(* IEC 61131-3 sources: pandora/pandora/aws-platform-main/aws-platform-main/src/WeldSystem/PowerSources, 5 files *)

(* ---- Pab.st ---- *)
USING Esab.Io;

NAMESPACE Esab.WeldSystem.PowerSources
    TYPE
        {S7.Extern=ReadWrite}
        PabData : STRUCT
            Input : PabToController;
            Output : ControllerToPab;
        END_STRUCT;

        // --- Interface struct declarations
        {S7.Extern=ReadWrite}
        PabToController : STRUCT
            /// Indicates that the Weld On command has been received.
            WeldStarted : DigitalInput;
            /// Set as soon as the welding requirements are met.
            Welding : DigitalInput;
            /// Indicates that the weld is finished. Only applicable for LAF/TAF.
            WeldingFinished : DigitalInput;
            /// TRUE when there is an error present that prohibits start.
            Error : DigitalInput;
            /// TRUE when it is possible to start a weld.
            ReadyToStart : DigitalInput;
            /// Indicates the currently selected weld method. TRUE = AC, FALSE = DC. Aristo 1000 only.
            WeldMethod : DigitalInput;
            /// Set when event information is available. Only set for ~5 seconds and then reset.
            Event : DigitalInput;
            /// Set when import or export function is active.
            FileBusy : DigitalInput;
            /// FALSE = Not coupled, TRUE = Coupled. If this is set the power source is master and has found its parallel slave(s).
            ParallelCoupleStatus : DigitalInput;
            /// The total number of errors or events detected. This equals the number of the last post in the error/event log.
            NumberOfErrors : UIntInput := (Endianness := Endianness#Big);
            /// Requested travel speed (cm/min).
            RequestedTravelSpeed : IntInput := (Endianness := Endianness#Little);
            /// The measured welding voltage.
            MeasuredVoltage : RealInput := (Endianness := Endianness#Little, Scale := REAL#0.1);
            /// The measured welding current.
            MeasuredCurrent : UIntInput := (Endianness := Endianness#Little);
            /// Measured wire speed (cm/min).
            MeasuredWireSpeed : IntInput := (Endianness := Endianness#Little);
            /// Measured travel speed (cm/min).
            MeasuredTravelSpeed : IntInput := (Endianness := Endianness#Little);
            /// The measured heat input.
            MeasuredHeatInput : RealInput := (Endianness := Endianness#Little, Scale := REAL#0.1);
            /// The currently set weld method. Aristo 1000 only.
            SetWeldMethod : UIntInput := (Endianness := Endianness#Big);
            /// The currently set regulation type. Aristo 1000 only.
            SetRegulationType : UIntInput := (Endianness := Endianness#Big);
            /// The AC frequency setpoint. Aristo 1000 only.
            SetAcFrequency : UIntInput := (Endianness := Endianness#Little);
            /// The AC balance setpoint. Aristo 1000 only.
            SetAcBalance : UIntInput := (Endianness := Endianness#Little);
            /// The voltage setpoint.
            SetVoltage : RealInput := (Endianness := Endianness#Little, Scale := REAL#0.1);
            /// The current setpoint.
            SetCurrent : UIntInput := (Endianness := Endianness#Little);
            /// Current wire speed setpoint (cm/min).
            SetWireSpeed : UIntInput := (Endianness := Endianness#Little);
            /// Current travel speed setpoint (cm/min).
            SetTravelSpeed : UIntInput := (Endianness := Endianness#Little);
            /// The current AC offset value.
            SetAcOffset : RealInput := (Endianness := Endianness#Little, Scale := REAL#0.1);
            /// The current AC phase shift value.
            SetAcPhaseShift : UIntInput := (Endianness := Endianness#Little);
            /// Requested wire speed (cm/min).
            RequestedWireSpeed : IntInput := (Endianness := Endianness#Little);
            /// Current weld data set
            SetWeldDataSet : UIntInput := (Endianness := Endianness#Little);
            ErrorEvent : ErrorEvent;
            /// Incremented at 2 Hz, when this value is incrementing the PAB can be considered alive and ready for communication.
            Heartbeat : UIntInput := (Endianness := Endianness#Little);
            /// The current start adjust value in %.
            SetStartAdjust : UIntInput := (Endianness := Endianness#Little);
            /// The current regulation dynamics value.
            SetRegulationDynamics : UIntInput := (Endianness := Endianness#Little);
            /// The current regulation inductance value.
            SetRegulationInductance : UIntInput := (Endianness := Endianness#Little);
        END_STRUCT;

        {S7.Extern=ReadWrite}
        ErrorEvent : STRUCT
            Code : WordInput := (Endianness := Endianness#Little);
            SubCode : UIntInput := (Endianness := Endianness#Big);
            NodeId : UIntInput := (Endianness := Endianness#Big);
            DeviceType : UIntInput := (Endianness := Endianness#Big);
            SubUnit : UIntInput := (Endianness := Endianness#Big);
        END_STRUCT;

        {S7.Extern=ReadWrite}
        ControllerToPab : STRUCT
            Common : PabInputCommon;
            InputArea : ARRAY[1..2] OF PabInputArea;
        END_STRUCT;

        {S7.Extern=ReadWrite}
        PabInputCommon : STRUCT
            /// Starts the weld when set to TRUE, to stop welding set this to FALSE.
            WeldOn : DigitalOutput;
            /// When this is set to TRUE the weld system will perform a quick stop (stopping without doing crater fill).
            QuickStop : DigitalOutput;
            /// Set to TRUE to jog the wire feed in the positive direction (down)
            WireFeedJogPos : DigitalOutput;
            /// Set to TRUE to jog the wire feed in the negative direction (up)
            WireFeedJogNeg : DigitalOutput;
            /// Set to TRUE to jog the travel axis in the positive direction
            TravelAxisJogPos : DigitalOutput;
            /// Set to TRUE to jog the travel axis in the negative direction
            TravelAxisJogNeg : DigitalOutput;
            /// Set to TRUE to jog the ICE wire feed in the positive direction (down)
            IceWireFeedJogPos : DigitalOutput;
            /// Set to TRUE to jog the ICE wire feed in the negative direction (up)
            IceWireFeedJogNeg : DigitalOutput;
            /// High speed (jogging)
            HighSpeed : DigitalOutput;
            /// Switches the active input area (0 = Input area #1, 1 = Input area #2)
            InputAreaSwitch : DigitalOutput;
            /// OPTIONAL! A heartbeat used to tell the PAB that the Controller is alive and well.
            Heartbeat : UIntOutput := (Endianness := Endianness#Big);
        END_STRUCT;

        {S7.Extern=ReadWrite}
        PabInputArea : STRUCT
            /// The weld method.
            WeldMethod : UIntOutput := (Endianness := Endianness#Big);
            /// The regulation type.
            RegulationType : UIntOutput := (Endianness := Endianness#Big);
            /// Weld voltage setpoint.
            Voltage : RealOutput := (Endianness := Endianness#Little, Scale := REAL#0.1);
            /// Wire speed setpoint (cm/min)
            WireSpeed : UIntOutput := (Endianness := Endianness#Little);
            /// Weld current setpoint
            Current : UIntOutput := (Endianness := Endianness#Little);
            /// Travel speed setpoint (cm/min)
            TravelSpeed : UIntOutput := (Endianness := Endianness#Little);
            /// AC frequency setpoint. Aristo 1000 only.
            AcFrequency : UIntOutput := (Endianness := Endianness#Little);
            /// AC balance setpoint. Aristo 1000 only
            AcBalance : UIntOutput := (Endianness := Endianness#Little);
            /// AC offset setpoint. Aristo 1000 only.
            AcOffset : RealOutput := (Endianness := Endianness#Little, Scale := REAL#0.1);
            /// AC phase shift setpoint. Aristo 1000 only
            AcPhaseShift : UIntOutput := (Endianness := Endianness#Little);
            /// Start adjust setpoint in %.
            StartAdjust : UIntOutput := (Endianness := Endianness#Little);
            /// Regulation dynamics setpoint.
            RegulationDynamics : UIntOutput := (Endianness := Endianness#Little);
            /// Regulation inductance setpoint.
            RegulationInductance : UIntOutput := (Endianness := Endianness#Little);
            /// ICE wire speed percentage.
            IceWireSpeedPercentage : UIntOutput := (Endianness := Endianness#Little);
        END_STRUCT;

        /// An enum representing the weld method
        WeldMethod : BYTE (
            DCp := BYTE#0,
            AC := BYTE#1,
            DCn := BYTE#2
        );

        RegulationType : BYTE (
            ConstantAmperage := BYTE#0,
            ConstantWire := BYTE#1,
            ConstantCurrent := BYTE#2
        );

        // --- I/O struct declarations
        {S7.Extern=ReadWrite}
        RawPabToController : STRUCT
            WeldStarted AT %X0.0 : BOOL;
            Welding AT %X0.1 : BOOL;
            WeldingFinished AT %X0.2 : BOOL;
            Error AT %X0.3 : BOOL;
            ReadyToStart AT %X1.3 : BOOL;
            WeldMethod AT %X2.2 : BOOL;
            Event AT %X2.4 : BOOL;
            FileBusy AT %X2.5 : BOOL;
            ParallelCoupleStatus AT %X2.7 : BOOL;
            NumberOfErrors AT %B4 : BYTE;
            RequestedTravelSpeed AT %B6 : INT;
            MeasuredVoltage AT %B8 : INT;
            MeasuredCurrent AT %B10 : UINT;
            MeasuredHeatInput AT %B12 : INT;
            MeasuredWireSpeed AT %B14 : INT;
            MeasuredTravelSpeed AT %B16 : INT;
            SetWeldMethod AT %B18 : BYTE;
            SetRegulationType AT %B19 : BYTE;
            SetAcFrequency AT %B20 : UINT;
            SetAcBalance AT %B22 : UINT;
            SetVoltage AT %B24 : UINT;
            SetCurrent AT %B26 : UINT;
            SetWireSpeed AT %B28 : UINT;
            SetTravelSpeed AT %B30 : UINT;
            SetAcOffset AT %B32 : INT;
            SetWeldDataSet AT %B34 : BYTE;
            SetAcPhaseShift AT %B36 : UINT;
            RequestedWireSpeed AT %B38 : INT;
            ErrorEvent AT %B40 : RawErrorEvent;
            Heartbeat AT %B46 : UINT;
            SetStartAdjust AT %B48 : UINT;
            SetRegulationDynamics AT %B50 : UINT;
            SetRegulationInductance AT %B52 : UINT;
        END_STRUCT;

        {S7.Extern=ReadWrite}
        RawErrorEvent : STRUCT
            Code AT %B0 : WORD;
            SubCode AT %B2 : BYTE;
            NodeId AT %B3 : BYTE;
            DeviceType AT %B4 : BYTE;
            SubUnit AT %B5 : BYTE;
        END_STRUCT;

        {S7.Extern=ReadWrite}
        RawControllerToPab : STRUCT
            Common AT %B0 : RawPabInputCommon;
            Area1 AT %B8 : RawPabInputArea;
            Area2 AT %B36 : RawPabInputArea;
        END_STRUCT;

        {S7.Extern=ReadWrite}
        RawPabInputCommon : STRUCT
            WeldOn AT %X0.0 : BOOL;
            QuickStop AT %X0.1 : BOOL;
            WireFeedJogPos AT %X0.4 : BOOL;
            WireFeedJogNeg AT %X0.5 : BOOL;
            TravelAxisJogPos AT %X0.6 : BOOL;
            TravelAxisJogNeg AT %X0.7 : BOOL;
            IceWireFeedJogPos AT %X1.0 : BOOL;
            IceWireFeedJogNeg AT %X1.1 : BOOL;
            HighSpeed AT %X1.2 : BOOL;
            InputAreaSwitch AT %X3.2 : BOOL;
            Heartbeat AT %B7 : BYTE;
        END_STRUCT;

        {S7.Extern=ReadWrite}
        RawPabInputArea : STRUCT
            WeldMethod AT %B0 : BYTE;
            RegulationType AT %B1 : BYTE;
            Voltage AT %B2 : UINT;
            WireSpeed AT %B4 : UINT;
            Current AT %B6 : UINT;
            TravelSpeed AT %B8 : UINT;
            AcFrequency AT %B10 : UINT;
            AcBalance AT %B12 : UINT;
            AcOffset AT %B14 : INT;
            AcPhaseShift AT %B16 : UINT;
            StartAdjust AT %B18 : UINT;
            RegulationDynamics AT %B20 : UINT;
            RegulationInductance AT %B22 : UINT;
            IceWireSpeedPercentage AT %B26 : UINT;
        END_STRUCT;
    END_TYPE

    FUNCTION PabRead
        VAR_INPUT
            Processed : REF_TO PabToController;
            Raw : REF_TO RawPabToController;
        END_VAR

        Processed^.WeldStarted.Read             (Raw^.WeldStarted);
        Processed^.Welding.Read                 (Raw^.Welding);
        Processed^.WeldingFinished.Read         (Raw^.WeldingFinished);
        Processed^.Error.Read                   (Raw^.Error);
        Processed^.ReadyToStart.Read            (Raw^.ReadyToStart);
        Processed^.WeldMethod.Read              (Raw^.WeldMethod);
        Processed^.Event.Read                   (Raw^.Event);
        Processed^.FileBusy.Read                (Raw^.FileBusy);
        Processed^.ParallelCoupleStatus.Read    (Raw^.ParallelCoupleStatus);
        Processed^.NumberOfErrors.Read          (Raw^.NumberOfErrors);
        Processed^.RequestedTravelSpeed.Read    (Raw^.RequestedTravelSpeed);
        Processed^.MeasuredVoltage.Read         (Raw^.MeasuredVoltage);
        Processed^.MeasuredCurrent.Read         (Raw^.MeasuredCurrent);
        Processed^.MeasuredHeatInput.Read       (Raw^.MeasuredHeatInput);
        Processed^.MeasuredWireSpeed.Read       (Raw^.MeasuredWireSpeed);
        Processed^.MeasuredTravelSpeed.Read     (Raw^.MeasuredTravelSpeed);
        Processed^.SetWeldMethod.Read           (Raw^.SetWeldMethod);
        Processed^.SetRegulationType.Read       (Raw^.SetRegulationType);
        Processed^.SetAcFrequency.Read          (Raw^.SetAcFrequency);
        Processed^.SetAcBalance.Read            (Raw^.SetAcBalance);
        Processed^.SetVoltage.Read              (Raw^.SetVoltage);
        Processed^.SetCurrent.Read              (Raw^.SetCurrent);
        Processed^.SetWireSpeed.Read            (Raw^.SetWireSpeed);
        Processed^.SetTravelSpeed.Read          (Raw^.SetTravelSpeed);
        Processed^.SetAcOffset.Read             (Raw^.SetAcOffset);
        Processed^.SetWeldDataSet.Read          (Raw^.SetWeldDataSet);
        Processed^.SetAcPhaseShift.Read         (Raw^.SetAcPhaseShift);
        Processed^.RequestedWireSpeed.Read      (Raw^.RequestedWireSpeed);
        Processed^.ErrorEvent.Code.Read         (Raw^.ErrorEvent.Code);
        Processed^.ErrorEvent.SubCode.Read      (Raw^.ErrorEvent.SubCode);
        Processed^.ErrorEvent.NodeId.Read       (Raw^.ErrorEvent.NodeId);
        Processed^.ErrorEvent.DeviceType.Read   (Raw^.ErrorEvent.DeviceType);
        Processed^.ErrorEvent.SubUnit.Read      (Raw^.ErrorEvent.SubUnit);
        Processed^.Heartbeat.Read               (Raw^.Heartbeat);
        Processed^.SetStartAdjust.Read          (Raw^.SetStartAdjust);
        Processed^.SetRegulationDynamics.Read   (Raw^.SetRegulationDynamics);
        Processed^.SetRegulationInductance.Read (Raw^.SetRegulationInductance);
    END_FUNCTION

    FUNCTION PabWrite
        VAR_INPUT
            Processed : REF_TO ControllerToPab;
            Raw : REF_TO RawControllerToPab;
        END_VAR

        Processed^.Common.WeldOn.Write              (Raw^.Common.WeldOn);
        Processed^.Common.QuickStop.Write           (Raw^.Common.QuickStop);
        Processed^.Common.Heartbeat.Write           (Raw^.Common.Heartbeat);
        Processed^.Common.WireFeedJogPos.Write      (Raw^.Common.WireFeedJogPos);
        Processed^.Common.WireFeedJogNeg.Write      (Raw^.Common.WireFeedJogNeg);
        Processed^.Common.TravelAxisJogPos.Write    (Raw^.Common.TravelAxisJogPos);
        Processed^.Common.TravelAxisJogNeg.Write    (Raw^.Common.TravelAxisJogNeg);
        Processed^.Common.IceWireFeedJogPos.Write   (Raw^.Common.IceWireFeedJogPos);
        Processed^.Common.IceWireFeedJogNeg.Write   (Raw^.Common.IceWireFeedJogNeg);
        Processed^.Common.HighSpeed.Write           (Raw^.Common.HighSpeed);
        Processed^.Common.InputAreaSwitch.Write     (Raw^.Common.InputAreaSwitch);

        Processed^.InputArea[1].WeldMethod.Write               (Raw^.Area1.WeldMethod);
        Processed^.InputArea[1].RegulationType.Write           (Raw^.Area1.RegulationType);
        Processed^.InputArea[1].Voltage.Write                  (Raw^.Area1.Voltage);
        Processed^.InputArea[1].WireSpeed.Write                (Raw^.Area1.WireSpeed);
        Processed^.InputArea[1].Current.Write                  (Raw^.Area1.Current);
        Processed^.InputArea[1].TravelSpeed.Write              (Raw^.Area1.TravelSpeed);
        Processed^.InputArea[1].AcFrequency.Write              (Raw^.Area1.AcFrequency);
        Processed^.InputArea[1].AcBalance.Write                (Raw^.Area1.AcBalance);
        Processed^.InputArea[1].AcOffset.Write                 (Raw^.Area1.AcOffset);
        Processed^.InputArea[1].AcPhaseShift.Write             (Raw^.Area1.AcPhaseShift);
        Processed^.InputArea[1].StartAdjust.Write              (Raw^.Area1.StartAdjust);
        Processed^.InputArea[1].RegulationDynamics.Write       (Raw^.Area1.RegulationDynamics);
        Processed^.InputArea[1].RegulationInductance.Write     (Raw^.Area1.RegulationInductance);
        Processed^.InputArea[1].IceWireSpeedPercentage.Write   (Raw^.Area1.IceWireSpeedPercentage);

        Processed^.InputArea[2].WeldMethod.Write               (Raw^.Area2.WeldMethod);
        Processed^.InputArea[2].RegulationType.Write           (Raw^.Area2.RegulationType);
        Processed^.InputArea[2].Voltage.Write                  (Raw^.Area2.Voltage);
        Processed^.InputArea[2].WireSpeed.Write                (Raw^.Area2.WireSpeed);
        Processed^.InputArea[2].Current.Write                  (Raw^.Area2.Current);
        Processed^.InputArea[2].TravelSpeed.Write              (Raw^.Area2.TravelSpeed);
        Processed^.InputArea[2].AcFrequency.Write              (Raw^.Area2.AcFrequency);
        Processed^.InputArea[2].AcBalance.Write                (Raw^.Area2.AcBalance);
        Processed^.InputArea[2].AcOffset.Write                 (Raw^.Area2.AcOffset);
        Processed^.InputArea[2].AcPhaseShift.Write             (Raw^.Area2.AcPhaseShift);
        Processed^.InputArea[2].StartAdjust.Write              (Raw^.Area2.StartAdjust);
        Processed^.InputArea[2].RegulationDynamics.Write       (Raw^.Area2.RegulationDynamics);
        Processed^.InputArea[2].RegulationInductance.Write     (Raw^.Area2.RegulationInductance);
        Processed^.InputArea[2].IceWireSpeedPercentage.Write   (Raw^.Area2.IceWireSpeedPercentage);
    END_FUNCTION

END_NAMESPACE

(* ---- PowerSource.st ---- *)
USING Esab.Utils.Assets;
USING Esab.Utils.Timer;
USING Esab.Utils.Io;

USING Esab.WeldSystem;

USING System.FastMath;

NAMESPACE Esab.WeldSystem.PowerSources

    INTERFACE IPowerSource
        /// Intended for cyclic execution
        METHOD Execute
        END_METHOD

        /// Sets a listener to this power source
        METHOD SetListener
            VAR_INPUT
                listener : IPowerSourceListener;
            END_VAR
        END_METHOD

        /// Initiates the welding sequence
        METHOD Start
        END_METHOD

        /// Stops the welding sequence in a controlled manner
        METHOD Stop
        END_METHOD

        /// Stops the welding sequence faster, skips the stop phase
        METHOD QuickStop
        END_METHOD

        /// Sets remote start towards the power source
        METHOD RemoteStart
        END_METHOD

        /// Sets remote stop towards the power source
        METHOD RemoteStop
        END_METHOD

        /// Returns a reference to the currently active input area
        METHOD ActiveArea : REF_TO SetPoints
        END_METHOD

        /// Returns a reference to the currently passive input area
        METHOD PassiveArea : REF_TO SetPoints
        END_METHOD

        /// Switch the active and passive areas
        METHOD SwitchActivePassive
        END_METHOD

        /// Sets the travel control (NOTE: Async)
        METHOD SetTravelControl
            VAR_INPUT
                control : TravelControl;
            END_VAR
        END_METHOD

        /// Sets the travel motor drive (NOTE: Async)
        METHOD SetTravelMotorDrive
            VAR_INPUT
                drive : TravelMotorDrive;
            END_VAR
        END_METHOD

        /// Sets the tandem role of this power source (NOTE: Async)
        METHOD SetTandemRole
            VAR_INPUT
                role : TandemRole;
            END_VAR
        END_METHOD

        /// Sets the start type (NOTE: Async)
        METHOD SetStartType
            VAR_INPUT
                startType : StartType;
            END_VAR
        END_METHOD

        /// Sets normal wire feed jog speed (NOTE: Async)
        METHOD SetWireFeedJogSpeed
            VAR_INPUT
                speed : UINT;
            END_VAR
        END_METHOD

        /// Sets wire feed jog high speed (NOTE: Async)
        METHOD SetWireFeedJogHighSpeed
            VAR_INPUT
                speed : UINT;
            END_VAR
        END_METHOD

        /// Applies a configuration to the wire motor
        /// Returns FALSE if it is not currently possible to set configuration
        METHOD ApplyWireMotorConfiguration : BOOL
            VAR_INPUT
                motorConfiguration : REF_TO MotorConfiguration;
            END_VAR
        END_METHOD

        /// ID of the power source
        METHOD GetId : UINT
        END_METHOD

        /// Node ID used by this power source
        METHOD GetNodeId : UINT
        END_METHOD

        /// The actual weld system type that is connected
        METHOD GetWeldSystemType : WeldSystemType
        END_METHOD

        /// Travel control (Off/Enabled)
        METHOD GetTravelControl : TravelControl
        END_METHOD

        /// Travel motor drive (Faa/External)
        METHOD GetTravelMotorDrive : TravelMotorDrive
        END_METHOD

        /// Tandem role (Head/Tail)
        METHOD GetTandemRole : TandemRole
        END_METHOD

        /// Returns TRUE if the welding system is welding
        METHOD IsWelding : BOOL
        END_METHOD

        /// Returns TRUE if the PLC has active communication with the PAB
        METHOD IsConnected : BOOL
        END_METHOD

        /// Returns TRUE if the power source reports as ready to start
        METHOD IsReadyToStart : BOOL
        END_METHOD

        /// Returns TRUE if the power source reports it has an error
        METHOD HasError : BOOL
        END_METHOD

        /// Returns the measured welding voltage.
        METHOD GetMeasuredVoltage : REAL
        END_METHOD

        /// Returns the measured wire speed (cm/min)
        METHOD GetMeasuredWireSpeed : INT
        END_METHOD

        /// Returns the measured travel speed (cm/min)
        METHOD GetMeasuredTravelSpeed : INT
        END_METHOD

        /// Returns the measured heat input (kJ/cm)
        METHOD GetMeasuredHeatInput : REAL
        END_METHOD

        /// Returns the currently set weld data set
        METHOD GetWeldDataSet : UINT
        END_METHOD

        /// Returns the requested (by the power source) travel speed
        METHOD GetRequestedTravelSpeed : INT
        END_METHOD

        /// Returns the requested (by the power source) wire speed
        METHOD GetRequestedWireSpeed : INT
        END_METHOD

        /// Returns TRUE if the node with the given ID is connected
        METHOD NodeIsConnected : BOOL
            VAR_INPUT
                nodeId : UINT;
            END_VAR
        END_METHOD

        /// Returns the information of the given node
        METHOD GetNodeInformation : NodeInformation
            VAR_INPUT
                nodeId : UINT;
            END_VAR
        END_METHOD

        METHOD WireFeedJogPos
            VAR_INPUT
                highSpeed : BOOL;
            END_VAR
        END_METHOD

        METHOD WireFeedJogNeg
            VAR_INPUT
                highSpeed : BOOL;
            END_VAR
        END_METHOD

        METHOD TravelAxisJogPos
            VAR_INPUT
                highSpeed : BOOL;
            END_VAR
        END_METHOD

        METHOD TravelAxisJogNeg
            VAR_INPUT
                highSpeed : BOOL;
            END_VAR
        END_METHOD

        /// Initiates a read of all connected nodes (unless already reading)
        METHOD ReadNodes
        END_METHOD

        METHOD WriteAsync
            VAR_INPUT
                record : DataRecord;
                value : UINT;
            END_VAR
        END_METHOD

        METHOD WriteAsync
            VAR_INPUT
                command: REF_TO UIntAsyncCommand;
            END_VAR
        END_METHOD

        METHOD ReadAsync
            VAR_INPUT
                record : DataRecord;
            END_VAR
        END_METHOD

        METHOD ReadAsync
            VAR_INPUT
                command: REF_TO UIntAsyncCommand;
            END_VAR
        END_METHOD
    END_INTERFACE

    INTERFACE IHeartBeat
        /// Returns TRUE if this object is initialized
        METHOD IsInitialized : BOOL
        END_METHOD

        /// Cyclic execution to evaluate heartbeat
        METHOD Execute
        END_METHOD

        /// Returns TRUE if a heartbeat is detected
        METHOD Alive : BOOL
        END_METHOD

        /// Returns TRUE if no heartbeat is detected
        METHOD Dead : BOOL
        END_METHOD
    END_INTERFACE

    CLASS Heartbeat IMPLEMENTS IHeartbeat
        VAR PUBLIC
            Input : IUIntInput;
            Timer: ITimer;
        END_VAR

        VAR PRIVATE
            _value : UINT;
            _lastValue : UINT;
            _alive : BOOL;
        END_VAR

        METHOD PUBLIC IsInitialized : BOOL
            IsInitialized := Input <> NULL AND Timer <> NULL;
        END_METHOD

        METHOD PUBLIC Execute
            IF NOT THIS.IsInitialized() THEN
                _alive := FALSE;
                RETURN;
            END_IF;

            _lastValue := _value;
            _value := Input.GetValue();

            Timer.Execute(_value = _lastValue, LT#10s);
            _alive := NOT Timer.Expired();
        END_METHOD

        METHOD PUBLIC Alive : BOOL
            Alive := _alive;
        END_METHOD

        METHOD PUBLIC Dead : BOOL
            Dead := NOT _alive;
        END_METHOD
    END_CLASS

    INTERFACE IPowerSourceListener
        /// Called when a power source becomes connected
        METHOD PowerSourceConnected
            VAR_INPUT
                /// The id (enumeration) of the power source
                id : UINT;
            END_VAR
        END_METHOD

        /// Called when a power source disconnects
        METHOD PowerSourceDisconnected
            VAR_INPUT
                /// The id (enumeration) of the power source
                id : UINT;
            END_VAR
        END_METHOD
    END_INTERFACE

    TYPE
        WeldProcess : INT(
            Saw := 0,
            Gmaw := 1,
            Gouging := 2
        );

        WireType : INT(
            FeSolidSingle := 0,
            FeSolidTwin := 1,
            FeTubeSingle := 2,
            FeTubeTwin := 3,
            SsSolidSingle := 4,
            SsSolidTwin := 5,
            SsTubeSingle := 6,
            SsTubeTwin := 7,
            AlSolidSingle := 8,
            AlSolidTwin := 9,
            StripSingle := 10,
            Gouging := 11
        );

        StartType : INT(
            Direct := 0,
            Scratch := 1,
            Lwas := 2,
            LwasMan := 3
        );

        TravelControl : INT(
            Off := 0,
            Enabled := 1
        );

        TravelMotorDrive : INT(
            Faa := 0,
            External := 1
        );

        TandemRole : INT(
            Head := 0,
            Slave := 1
        );

        /// Container for values read from async commands
        StatusBuffer : STRUCT
            /// Node ID used by this power source
            NodeId : UINT;
            /// The actual weld system type that is connected
            WeldSystemType : WeldSystemType;
            /// Travel control (Off/Enabled)
            TravelControl : TravelControl;
            /// Travel motor drive (Faa/External)
            TravelMotorDrive : TravelMotorDrive;
            /// Tandem role (Head/Tail)
            TandemRole : TandemRole;
        END_STRUCT;
    END_TYPE

    CLASS PowerSourceObservable IMPLEMENTS IAssetObservable
        VAR PUBLIC
            State : PowerSourceState;
            ReadyToStart : BOOL;
            Welding : BOOL;
            Error : BOOL;
            Connected : BOOL;
            WeldMethod : WeldMethod;
            MeasuredVoltage : REAL;
            MeasuredCurrent : UINT;
            MeasuredHeatInput : REAL;
            MeasuredWireSpeed : INT;
            MeasuredTravelSpeed : INT;
            RequestedWireSpeed : INT;
            RequestedTravelSpeed : INT;
            SetPoints : SetPoints;
        END_VAR
    END_CLASS

    FUNCTION CalculateMotorScaleFactors
        VAR_INPUT
            motorConfiguration : REF_TO MotorConfiguration;
        END_VAR

        VAR_OUTPUT
            nominator : UINT;
            denominator : UINT;
        END_VAR

        nominator := TO_UINT(TO_LREAL(motorConfiguration^.Gear.N2) / motorConfiguration^.Gear.N1 * motorConfiguration^.Rpm * motorConfiguration^.FeedRollDiameter * Constants#PI);
        denominator := TO_UINT(TO_UDINT(motorConfiguration^.Rpm) * motorConfiguration^.EncoderPpr / UINT#60);
    END_FUNCTION

    TYPE
        {S7.Extern=ReadWrite}
        RuntimeParameters : STRUCT
            WireFeedJogSpeed : UINT;
            WireFeedJogHighSpeed : UINT;
        END_STRUCT;

        {S7.Extern=ReadWrite}
        HardwareConfiguration : STRUCT
            WireMotor : MotorConfiguration;
        END_STRUCT;

        {S7.Extern=ReadWrite}
        MotorConfiguration : STRUCT
            Gear : Gear;
            Rpm : UINT;
            FeedRollDiameter : UINT;
            EncoderPpr : UINT;
            MaxCurrent : UINT;
        END_STRUCT;

        {S7.Extern=ReadWrite}
        Gear : STRUCT
            N1 : UINT;
            N2 : UINT;
        END_STRUCT;

        {S7.Extern=ReadWrite}
        Io : STRUCT
            Pab : PabData;
            Output : Output;
        END_STRUCT;

        {S7.Extern=ReadWrite}
        Output : STRUCT
            RemoteStart : DigitalOutput;
        END_STRUCT;

        PowerSourceState : INT(
            Idle := 0,
            NotConnected := 1,
            Error := 2,
            Welding := 3
        );

        SetPoints : STRUCT
            Voltage : REAL;
            Current : UINT;
            WireSpeed : UINT;
            TravelSpeed : UINT;
            AcFrequency : UINT;
            AcBalance : UINT;
            AcOffset : REAL;
            AcPhaseShift : UINT;
            WeldMethod : WeldMethod;
            RegulationType : RegulationType;
            StartAdjust : UINT;
            RegulationDynamics : UINT;
            RegulationInductance : UINT;
            IceWireSpeedPercentage : UINT;
        END_STRUCT;
    END_TYPE

END_NAMESPACE

(* ---- Aristo1000.st ---- *)
USING Esab.Api;
USING Esab.Utils.Alarming;
USING Esab.Utils;
USING Esab.Utils.Assets;
USING Esab.WeldSystem.PowerSources;
USING Esab.Utils.Alarming;
USING Siemens.Simatic.S71500.Alarming;
USING Siemens.Simatic.S71500.DistributedIO;

NAMESPACE Esab.WeldSystem.PowerSources.Aristo1000

    /// This class implements an Aristo 1000 power source
    CLASS PowerSource EXTENDS Asset IMPLEMENTS IPowerSource, IAsyncCommandListener
        VAR PRIVATE
            _id : UINT;
            _ioDeviceId : WORD;
            _heartbeat: IHeartBeat;
            _io : REF_TO Io;
            _runtimeParameters : REF_TO RuntimeParameters;
            _hardwareConfiguration : REF_TO HardwareConfiguration;
            _asyncInterface : IAsyncInterface;
            _asyncCommands : AsyncCommands;
            _errorAlarm : IAlarm;
            _heartbeatAlarm : IAlarm;
            _asyncCommandReadAlarm : IAlarm;
            _asyncCommandWriteAlarm : IAlarm;
            _asyncCommandNullAlarm : IAlarm;

            _readingNodes : BOOL := FALSE;
            _currentlyReadingNodeId : UINT := UINT#0;
            _nodeInformation : ARRAY [1..31] OF NodeInformation;
            _observable : PowerSourceObservable;
            _listener : IPowerSourceListener := NULL;
            _isConnected : BOOL := FALSE;

            _nodeId : UINT := UINT#0;
            _weldSystemType : WeldSystemType;
            _travelControl : TravelControl;
            _travelMotorDrive : TravelMotorDrive;
            _tandemRole : TandemRole;
            _inputAreaSwitch : BOOL := FALSE; // Area 2 is active if True
            _inputArea : ARRAY [1..2] OF SetPoints;

            // Commands used when reading/writing custom records
            _writeUIntAsyncCommand : UIntAsyncCommand;
            _readUIntAsyncCommand : UIntAsyncCommand;

            _highSpeed : BOOL := FALSE;
            _wireFeedJogPos : BOOL := FALSE;
            _wireFeedJogNeg : BOOL := FALSE;
            _travelAxisJogPos : BOOL := FALSE;
            _travelAxisJogNeg : BOOL := FALSE;
        END_VAR

        METHOD PUBLIC Setup
            VAR_INPUT
                id : UINT;
                ioDeviceId : WORD;
                heartbeat: IHeartBeat;
                io : REF_TO Io;
                runtimeParameters : REF_TO RuntimeParameters;
                hardwareConfiguration : REF_TO HardwareConfiguration;
                asyncInterface : IAsyncInterface;
                errorAlarm : IAlarm;
                heartbeatAlarm : IAlarm;
                asyncCommandReadAlarm : IAlarm;
                asyncCommandWriteAlarm : IAlarm;
                asyncCommandNullAlarm : IAlarm;
                setupAlarm : IAlarm;
            END_VAR

            _id := id;
            _ioDeviceId := ioDeviceId;
            _heartbeat := heartbeat;
            _io := io;
            _runtimeParameters := runtimeParameters;
            _hardwareConfiguration := hardwareConfiguration;
            _asyncInterface := asyncInterface;
            _asyncInterface.SetListener(THIS);
            _errorAlarm := errorAlarm;
            _heartbeatAlarm := heartbeatAlarm;
            _asyncCommandReadAlarm := asyncCommandReadAlarm;
            _asyncCommandWriteAlarm := asyncCommandWriteAlarm;
            _asyncCommandNullAlarm := asyncCommandNullAlarm;
            _setupAlarm := setupAlarm;

            _isSetup := _io <> NULL AND
                        _heartbeat <> NULL AND
                        _runtimeParameters <> NULL AND
                        _hardwareConfiguration <> NULL AND
                        _errorAlarm <> NULL AND
                        _heartbeatAlarm <> NULL AND
                        _asyncCommandReadAlarm <> NULL AND
                        _asyncCommandWriteAlarm <> NULL AND
                        _asyncCommandNullAlarm <> NULL;

            IF _isSetup THEN
                THIS.WriteAsync(DataRecord#WireJogLowSpeed, _runtimeParameters^.WireFeedJogSpeed);
                THIS.WriteAsync(DataRecord#WireJogHighSpeed, _runtimeParameters^.WireFeedJogHighSpeed);
            END_IF;
        END_METHOD

        METHOD PUBLIC OVERRIDE Execute
            SUPER.Execute();

            IF _setupAlarm.IsActive() THEN
                RETURN;
            END_IF;

            _heartbeat.Execute();

            _heartbeatAlarm.Execute(SIG := _heartbeat.Dead());

            IF _heartbeat.Dead() THEN
                IF _isConnected AND _listener <> NULL THEN
                    _listener.PowerSourceDisconnected(THIS.GetId());
                END_IF;

                RETURN;
            ELSIF NOT _isConnected AND _listener <> NULL THEN
                THIS.ReadNodes();
                _listener.PowerSourceConnected(THIS.GetId());
            END_IF;

            _isConnected := _heartbeat.Alive();

            THIS.SetHeartbeat(THIS.GetHeartbeat());

            _errorAlarm.Execute(SIG := _io^.Pab.Input.Error.GetValue());

            _io^.Pab.Output.Common.HighSpeed.SetValue(_highSpeed);
            _io^.Pab.Output.Common.WireFeedJogPos.SetValue(_wireFeedJogPos);
            _io^.Pab.Output.Common.WireFeedJogNeg.SetValue(_wireFeedJogNeg);
            _io^.Pab.Output.Common.TravelAxisJogPos.SetValue(_travelAxisJogPos);
            _io^.Pab.Output.Common.TravelAxisJogNeg.SetValue(_travelAxisJogNeg);

            _highSpeed := FALSE;
            _wireFeedJogPos := FALSE;
            _wireFeedJogNeg := FALSE;
            _travelAxisJogPos := FALSE;
            _travelAxisJogNeg := FALSE;

            IF _io^.Pab.Input.Welding.FallingEdge() THEN
                THIS.Stop();
            END_IF;

            _asyncInterface.Execute();

            THIS.UpdateObservable();
            THIS.UpdateSetpoints();
        END_METHOD

        METHOD PUBLIC OVERRIDE UpdateState
            IF _setupAlarm.IsActive() THEN
                _currentState := PowerSourceState#Error;
            ELSIF NOT THIS.IsConnected() THEN
                _currentState := PowerSourceState#NotConnected;
            ELSIF THIS.IsWelding() THEN
                _currentState := PowerSourceState#Welding;
            ELSIF _errorAlarm.IsActive() OR _asyncCommandReadAlarm.IsActive() OR _asyncCommandWriteAlarm.IsActive() OR _asyncCommandNullAlarm.IsActive() THEN
                _currentState := PowerSourceState#Error;
            ELSE
                _currentState := PowerSourceState#Idle;
            END_IF;
        END_METHOD

        METHOD PUBLIC SetListener
            VAR_INPUT
                listener : IPowerSourceListener;
            END_VAR

            _listener := listener;
        END_METHOD

        METHOD PUBLIC Start
            _io^.Pab.Output.Common.WeldOn.SetValue(TRUE);
        END_METHOD

        METHOD PUBLIC Stop
            _io^.Pab.Output.Common.WeldOn.SetValue(FALSE);
        END_METHOD

        METHOD PUBLIC QuickStop
            _io^.Pab.Output.Common.WeldOn.SetValue(FALSE);
            _io^.Pab.Output.Common.QuickStop.SetValue(TRUE);
        END_METHOD

        METHOD PUBLIC RemoteStart
            _io^.Output.RemoteStart.SetValue(TRUE);
        END_METHOD

        METHOD PUBLIC RemoteStop
            _io^.Output.RemoteStart.SetValue(FALSE);
        END_METHOD

        METHOD PUBLIC ActiveArea : REF_TO SetPoints
            IF NOT _inputAreaSwitch THEN
                ActiveArea := REF(_inputArea[1]);
            ELSE
                ActiveArea := REF(_inputArea[2]);
            END_IF;
        END_METHOD

        METHOD PUBLIC PassiveArea : REF_TO SetPoints
            IF NOT _inputAreaSwitch THEN
                PassiveArea := REF(_inputArea[2]);
            ELSE
                PassiveArea := REF(_inputArea[1]);
            END_IF;
        END_METHOD

        METHOD PUBLIC SwitchActivePassive
            _inputAreaSwitch := NOT _inputAreaSwitch;
            _io^.Pab.Output.Common.InputAreaSwitch.SetValue(_inputAreaSwitch);
        END_METHOD

        METHOD PUBLIC IsWelding : BOOL
            IsWelding := _io^.Pab.Input.Welding.GetValue() OR _io^.Pab.Input.WeldStarted.GetValue();
        END_METHOD

        METHOD PUBLIC IsConnected : BOOL
            IsConnected := _heartbeat.Alive();
        END_METHOD

        METHOD PUBLIC IsReadyToStart : BOOL
            IsReadyToStart := _io^.Pab.Input.ReadyToStart.GetValue();
        END_METHOD

        METHOD PUBLIC HasError : BOOL
            HasError := _io^.Pab.Input.Error.GetValue();
        END_METHOD

        METHOD PUBLIC SetTravelControl
            VAR_INPUT
                control : TravelControl;
            END_VAR

            _travelControl := control;
            _asyncCommands.TravelControl.Value := TO_UINT(control);

            _asyncInterface.WriteCommand(REF(_asyncCommands.TravelControl));
        END_METHOD

        METHOD PUBLIC SetTravelMotorDrive
            VAR_INPUT
                drive : TravelMotorDrive;
            END_VAR

            _travelMotorDrive := drive;
            _asyncCommands.TravelMotorDrive.Value := TO_UINT(drive);

            _asyncInterface.WriteCommand(REF(_asyncCommands.TravelMotorDrive));
        END_METHOD

        METHOD PUBLIC SetTandemRole
            VAR_INPUT
                role : TandemRole;
            END_VAR

            _tandemRole := role;
            _asyncCommands.TandemRole.Value := TO_UINT(role);

            _asyncInterface.WriteCommand(REF(_asyncCommands.TandemRole));
        END_METHOD

        METHOD PUBLIC SetStartType
            VAR_INPUT
                startType : StartType;
            END_VAR

            _asyncCommands.StartType.Value := TO_UINT(startType);

            _asyncInterface.WriteCommand(REF(_asyncCommands.StartType));
        END_METHOD

        METHOD PUBLIC SetWireFeedJogSpeed
            VAR_INPUT
                speed : UINT;
            END_VAR

            _asyncCommands.JogWireFeedSpeed.Value := speed;
            _asyncInterface.WriteCommand(REF(_asyncCommands.JogWireFeedSpeed));
        END_METHOD

        METHOD PUBLIC SetWireFeedJogHighSpeed
            VAR_INPUT
                speed : UINT;
            END_VAR

            _asyncCommands.JogWireFeedHighSpeed.Value := speed;
            _asyncInterface.WriteCommand(REF(_asyncCommands.JogWireFeedHighSpeed));
        END_METHOD

        METHOD PUBLIC GetId : UINT
            GetId := _id;
        END_METHOD

        METHOD PUBLIC GetNodeId : UINT
            GetNodeId := _nodeId;
        END_METHOD

        METHOD PUBLIC GetWeldSystemType : WeldSystemType
            GetWeldSystemType := _weldSystemType;
        END_METHOD

        METHOD PUBLIC GetTravelControl : TravelControl
            GetTravelControl := _travelControl;
        END_METHOD

        METHOD PUBLIC GetTravelMotorDrive : TravelMotorDrive
            GetTravelMotorDrive := _travelMotorDrive;
        END_METHOD

        METHOD PUBLIC GetTandemRole : TandemRole
            GetTandemRole := _tandemRole;
        END_METHOD

        METHOD PUBLIC GetMeasuredVoltage : REAL
            GetMeasuredVoltage := _io^.Pab.Input.MeasuredVoltage.GetValue();
        END_METHOD

        METHOD PUBLIC GetMeasuredCurrent : UINT
            GetMeasuredCurrent := _io^.Pab.Input.MeasuredCurrent.GetValue();
        END_METHOD

        METHOD PUBLIC GetMeasuredWireSpeed : INT
            GetMeasuredWireSpeed := _io^.Pab.Input.MeasuredWireSpeed.GetValue();
        END_METHOD

        METHOD PUBLIC GetMeasuredTravelSpeed : INT
            GetMeasuredTravelSpeed := _io^.Pab.Input.MeasuredTravelSpeed.GetValue();
        END_METHOD

        METHOD PUBLIC GetMeasuredHeatInput : REAL
            GetMeasuredHeatInput := _io^.Pab.Input.MeasuredHeatInput.GetValue();
        END_METHOD

        METHOD PUBLIC GetWeldDataSet : UINT
            GetWeldDataSet := _io^.Pab.Input.SetWeldDataSet.GetValue();
        END_METHOD

        METHOD PUBLIC GetRequestedTravelSpeed : INT
            GetRequestedTravelSpeed := _io^.Pab.Input.RequestedTravelSpeed.GetValue();
        END_METHOD

        METHOD PUBLIC GetRequestedWireSpeed : INT
            GetRequestedWireSpeed := _io^.Pab.Input.RequestedWireSpeed.GetValue();
        END_METHOD

        METHOD PUBLIC WireFeedJogPos
            VAR_INPUT
                highSpeed : BOOL;
            END_VAR

            _highSpeed := highSpeed;
            _wireFeedJogPos := TRUE;
        END_METHOD

        METHOD PUBLIC WireFeedJogNeg
            VAR_INPUT
                highSpeed : BOOL;
            END_VAR

            _highSpeed := highSpeed;
            _wireFeedJogNeg := TRUE;
        END_METHOD

        METHOD PUBLIC TravelAxisJogPos
            VAR_INPUT
                highSpeed : BOOL;
            END_VAR

            _highSpeed := highSpeed;
            _travelAxisJogPos := TRUE;
        END_METHOD

        METHOD PUBLIC TravelAxisJogNeg
            VAR_INPUT
                highSpeed : BOOL;
            END_VAR

            _highSpeed := highSpeed;
            _travelAxisJogNeg := TRUE;
        END_METHOD

        METHOD PUBLIC ReadNodes
            IF _readingNodes = FALSE THEN
                _readingNodes := TRUE;
                _asyncInterface.ReadCommand(REF(_asyncCommands.ConnectedUnits));
            END_IF;
        END_METHOD

        METHOD PUBLIC NodeIsConnected : BOOL
            VAR_INPUT
                nodeId : UINT;
            END_VAR

            NodeIsConnected := _nodeInformation[nodeId].Connected;
        END_METHOD

        METHOD PUBLIC GetNodeInformation : NodeInformation
            VAR_INPUT
                nodeId : UINT;
            END_VAR

            GetNodeInformation := _nodeInformation[nodeId];
        END_METHOD

        METHOD PUBLIC ApplyWireMotorConfiguration : BOOL
            VAR_INPUT
                motorConfiguration : REF_TO MotorConfiguration;
            END_VAR

            VAR_TEMP
                _scaleFactor1 : UINT;
                _scaleFactor2 : UINT;
            END_VAR

            IF motorConfiguration = NULL THEN
                ApplyWireMotorConfiguration := FALSE;
                RETURN;
            END_IF;

            IF NOT THIS.IsWelding() THEN
                CalculateMotorScaleFactors(motorConfiguration, _scaleFactor1, _scaleFactor2);

                _asyncCommands.WireMotorScaleFactor1.Value := _scaleFactor1;
                _asyncInterface.WriteCommand(REF(_asyncCommands.WireMotorScaleFactor1));

                _asyncCommands.WireMotorScaleFactor2.Value := _scaleFactor2;
                _asyncInterface.WriteCommand(REF(_asyncCommands.WireMotorScaleFactor2));

                _asyncCommands.MaxWireMotorCurrent.Value := motorConfiguration^.MaxCurrent;
                _asyncInterface.WriteCommand(REF(_asyncCommands.MaxWireMotorCurrent));
            ELSE
                ApplyWireMotorConfiguration := FALSE;
                RETURN;
            END_IF;

            ApplyWireMotorConfiguration := TRUE;
        END_METHOD

        METHOD PUBLIC WriteAsync
            VAR_INPUT
                record : DataRecord;
                value : UINT;
            END_VAR

            _writeUIntAsyncCommand.Index := record;
            _writeUIntAsyncCommand.Value := value;
            _asyncInterface.WriteCommand(REF(_writeUIntAsyncCommand));
        END_METHOD

        METHOD PUBLIC WriteAsync
            VAR_INPUT
                command: REF_TO UIntAsyncCommand;
            END_VAR

            _asyncInterface.WriteCommand(command);
        END_METHOD

        METHOD PUBLIC ReadAsync
            VAR_INPUT
                record : DataRecord;
            END_VAR

            _readUIntAsyncCommand.Index := record;
            _asyncInterface.ReadCommand(REF(_readUIntAsyncCommand));
        END_METHOD

        // For extrernal callers
        METHOD PUBLIC ReadAsync
            VAR_INPUT
                command: REF_TO UIntAsyncCommand;
            END_VAR
            _asyncInterface.ReadCommand(command);
        END_METHOD

        METHOD PUBLIC AsyncCommandCallback
            VAR_INPUT
                command : REF_TO AsyncCommand;
                status : CommandStatus;
            END_VAR

            VAR_TEMP
                _uintCommand : REF_TO UIntAsyncCommand;
                _udintCommand : REF_TO UDIntAsyncCommand;
                _nodeInfoCommand : REF_TO NodeInformationAsyncCommand;

                _index : UINT := UINT#0;
            END_VAR

            _asyncCommandNullAlarm.Execute(SIG := command = NULL);

            IF command = NULL THEN
                RETURN;
            END_IF;

            _asyncCommandReadAlarm.Execute(SIG := command^.GetType() = CommandType#Read && status = CommandStatus#Error, SD_1 := pass(command^.GetIndex()));
            _asyncCommandWriteAlarm.Execute(SIG := command^.GetType() = CommandType#Write && status = CommandStatus#Error, SD_1 := pass(command^.GetIndex()));

            IF command^.GetType() = CommandType#Write AND status = CommandStatus#Success THEN
                _asyncInterface.ReadCommand(command);
            ELSIF command^.GetType() = CommandType#Read THEN
                _uintCommand ?= command;
                _udintCommand ?= command;
                _nodeInfoCommand ?= command;

                CASE command^.Index OF
                    DataRecord#TravelControl:
                        IF _uintCommand <> NULL AND status = CommandStatus#Success THEN
                            _travelControl := TO_INT(_uintCommand^.Value);
                        END_IF;
                    DataRecord#TravelMotorDrive:
                        IF _uintCommand <> NULL AND status = CommandStatus#Success THEN
                            _travelMotorDrive := TO_INT(_uintCommand^.Value);
                        END_IF;
                    DataRecord#TandemRole:
                        IF _uintCommand <> NULL AND status = CommandStatus#Success THEN
                            _tandemRole := TO_INT(_uintCommand^.Value);
                        END_IF;
                    DataRecord#ConnectedUnits:
                        IF _udintCommand <> NULL AND status = CommandStatus#Success THEN
                            FOR _index := 1 TO UINT#31 DO
                                _nodeInformation[_index].Connected := ((SHR(TO_DWORD(_udintCommand^.Value), _index) & DWORD#1) <> DWORD#0);
                            END_FOR;

                            // This will kick off the reading of all nodes information
                            THIS.ReadNextConnectedNode();
                        END_IF;
                    DataRecord#NodeInformation:
                        IF _nodeInfoCommand <> NULL AND status = CommandStatus#Success THEN
                            _nodeInformation[_nodeInfoCommand^.Id].Version := _nodeInfoCommand^.Value.Version;
                            _nodeInformation[_nodeInfoCommand^.Id].SubVersion := _nodeInfoCommand^.Value.SubVersion;
                            _nodeInformation[_nodeInfoCommand^.Id].DeviceType := _nodeInfoCommand^.Value.DeviceType;
                            _nodeInformation[_nodeInfoCommand^.Id].MachineId := _nodeInfoCommand^.Value.MachineId;
                            IF _readingNodes THEN
                                THIS.ReadNextConnectedNode();
                            END_IF;
                        ELSE
                            THIS.CancelNodeReading();
                        END_IF;
                    DataRecord#Can2NodeId:
                        IF _uintCommand <> NULL THEN
                            _nodeId := _uintCommand^.Value;
                        END_IF;
                    DataRecord#GetWeldingSystem:
                        IF _uintCommand <> NULL THEN
                            _weldSystemType := _uintCommand^.Value;
                        END_IF;
                    DataRecord#WireJogLowSpeed:
                        if _uintCommand <> NULL THEN
                            IF _runtimeParameters <> NULL THEN
                                _runtimeParameters^.WireFeedJogSpeed := _uintCommand^.Value;
                            END_IF;
                        END_IF;
                    DataRecord#WireJogHighSpeed:
                        if _uintCommand <> NULL THEN
                            IF _runtimeParameters <> NULL THEN
                                _runtimeParameters^.WireFeedJogHighSpeed := _uintCommand^.Value;
                            END_IF;
                        END_IF;
                END_CASE;
            END_IF;
        END_METHOD

        METHOD PUBLIC OVERRIDE Observe : IAssetObservable
            Observe := _observable;
        END_METHOD

        METHOD PRIVATE SetHeartbeat
            VAR_INPUT
                value : UINT;
            END_VAR

            _io^.Pab.Output.Common.Heartbeat.SetValue(value);
        END_METHOD

        METHOD PRIVATE GetHeartbeat : UINT
            GetHeartbeat := _io^.Pab.Input.Heartbeat.GetValue();
        END_METHOD

        METHOD PRIVATE ReadNextConnectedNode
            VAR_TEMP
                isConnected : BOOL := FALSE;
            END_VAR

            _currentlyReadingNodeId := _currentlyReadingNodeId + UINT#1;

            WHILE _currentlyReadingNodeId <= UINT#31 AND NOT isConnected DO
                isConnected := _nodeInformation[_currentlyReadingNodeId].Connected;
                IF NOT isConnected THEN
                    _currentlyReadingNodeId := _currentlyReadingNodeId + UINT#1;
                END_IF;
            END_WHILE;

            IF _currentlyReadingNodeId <= UINT#31 THEN
                _asyncCommands.NodeInformation.Id := _currentlyReadingNodeId;
                _asyncInterface.WriteCommand(REF(_asyncCommands.NodeInformation));
            ELSE
                THIS.CancelNodeReading();
            END_IF;
        END_METHOD

        METHOD PRIVATE CancelNodeReading
            _currentlyReadingNodeId := UINT#0;
            _readingNodes := FALSE;
        END_METHOD

        METHOD PRIVATE UpdateObservable
            _observable.State := _currentState;
            _observable.ReadyToStart := THIS.IsReadyToStart();
            _observable.Error := THIS.HasError();
            _observable.Welding := THIS.IsWelding();
            _observable.Connected := THIS.IsConnected();
            _observable.MeasuredVoltage := THIS.GetMeasuredVoltage();
            _observable.MeasuredCurrent := THIS.GetMeasuredCurrent();
            _observable.MeasuredWireSpeed := THIS.GetMeasuredWireSpeed();
            _observable.MeasuredTravelSpeed := THIS.GetMeasuredTravelSpeed();
            _observable.MeasuredHeatInput := THIS.GetMeasuredHeatInput();
            _observable.RequestedWireSpeed := THIS.GetRequestedWireSpeed();
            _observable.RequestedTravelSpeed := THIS.GetRequestedTravelSpeed();
            _observable.SetPoints.Voltage := _io^.Pab.Input.SetVoltage.GetValue();
            _observable.SetPoints.Current := _io^.Pab.Input.SetCurrent.GetValue();
            _observable.SetPoints.WireSpeed := _io^.Pab.Input.SetWireSpeed.GetValue();
            _observable.SetPoints.TravelSpeed := _io^.Pab.Input.SetTravelSpeed.GetValue();
            _observable.SetPoints.AcFrequency := _io^.Pab.Input.SetAcFrequency.GetValue();
            _observable.SetPoints.AcBalance := _io^.Pab.Input.SetAcBalance.GetValue();
            _observable.SetPoints.AcOffset := _io^.Pab.Input.SetAcOffset.GetValue();
            _observable.SetPoints.AcPhaseShift := _io^.Pab.Input.SetAcPhaseShift.GetValue();
            _observable.SetPoints.WeldMethod := TO_BYTE(_io^.Pab.Input.SetWeldMethod.GetValue());
            _observable.SetPoints.RegulationType := TO_BYTE(_io^.Pab.Input.SetRegulationType.GetValue());
            _observable.SetPoints.StartAdjust := _io^.Pab.Input.SetStartAdjust.GetValue();
            _observable.SetPoints.RegulationDynamics := _io^.Pab.Input.SetRegulationDynamics.GetValue();
            _observable.SetPoints.RegulationInductance := _io^.Pab.Input.SetRegulationInductance.GetValue();
            // _observable.SetPoints.IceWireSpeedPercentage := _io^.Pab.Input.SetIceWireSpeedPercentage.GetValue(); // Not available
        END_METHOD

        METHOD PRIVATE UpdateSetpoints
            VAR_TEMP
                area1 : REF_TO SetPoints;
                area2 : REF_TO SetPoints;
            END_VAR

            IF NOT _inputAreaSwitch THEN
                area1 := THIS.ActiveArea();
                area2 := THIS.PassiveArea();
            ELSE
                area1 := THIS.PassiveArea();
                area2 := THIS.ActiveArea();
            END_IF;

            _io^.Pab.Output.InputArea[1].Voltage.SetValue(area1^.Voltage);
            _io^.Pab.Output.InputArea[1].Current.SetValue(area1^.Current);
            _io^.Pab.Output.InputArea[1].WireSpeed.SetValue(area1^.WireSpeed);
            _io^.Pab.Output.InputArea[1].TravelSpeed.SetValue(area1^.TravelSpeed);
            _io^.Pab.Output.InputArea[1].AcFrequency.SetValue(area1^.AcFrequency);
            _io^.Pab.Output.InputArea[1].AcBalance.SetValue(area1^.AcBalance);
            _io^.Pab.Output.InputArea[1].AcOffset.SetValue(area1^.AcOffset);
            _io^.Pab.Output.InputArea[1].AcPhaseShift.SetValue(area1^.AcPhaseShift);
            _io^.Pab.Output.InputArea[1].WeldMethod.SetValue(area1^.WeldMethod);
            _io^.Pab.Output.InputArea[1].RegulationType.SetValue(area1^.RegulationType);
            _io^.Pab.Output.InputArea[1].StartAdjust.SetValue(area1^.StartAdjust);
            _io^.Pab.Output.InputArea[1].RegulationDynamics.SetValue(area1^.RegulationDynamics);
            _io^.Pab.Output.InputArea[1].RegulationInductance.SetValue(area1^.RegulationInductance);
            _io^.Pab.Output.InputArea[1].IceWireSpeedPercentage.SetValue(area1^.IceWireSpeedPercentage);

            _io^.Pab.Output.InputArea[2].Voltage.SetValue(area2^.Voltage);
            _io^.Pab.Output.InputArea[2].Current.SetValue(area2^.Current);
            _io^.Pab.Output.InputArea[2].WireSpeed.SetValue(area2^.WireSpeed);
            _io^.Pab.Output.InputArea[2].TravelSpeed.SetValue(area2^.TravelSpeed);
            _io^.Pab.Output.InputArea[2].AcFrequency.SetValue(area2^.AcFrequency);
            _io^.Pab.Output.InputArea[2].AcBalance.SetValue(area2^.AcBalance);
            _io^.Pab.Output.InputArea[2].AcOffset.SetValue(area2^.AcOffset);
            _io^.Pab.Output.InputArea[2].AcPhaseShift.SetValue(area2^.AcPhaseShift);
            _io^.Pab.Output.InputArea[2].WeldMethod.SetValue(area2^.WeldMethod);
            _io^.Pab.Output.InputArea[2].RegulationType.SetValue(area2^.RegulationType);
            _io^.Pab.Output.InputArea[2].StartAdjust.SetValue(area2^.StartAdjust);
            _io^.Pab.Output.InputArea[2].RegulationDynamics.SetValue(area2^.RegulationDynamics);
            _io^.Pab.Output.InputArea[2].RegulationInductance.SetValue(area2^.RegulationInductance);
            _io^.Pab.Output.InputArea[2].IceWireSpeedPercentage.SetValue(area2^.IceWireSpeedPercentage);
        END_METHOD
    END_CLASS

END_NAMESPACE

(* ---- AsyncCommands.st ---- *)
USING Esab.Io;
USING Esab.Utils.Collections;

NAMESPACE Esab.WeldSystem.PowerSources

    CLASS AsyncCommands
        VAR PUBLIC
            WireType : UIntAsyncCommand := (Index := DataRecord#WeldMethod);
            WireDimension : UIntAsyncCommand := (Index := DataRecord#WeldMethod);
            StartType : UIntAsyncCommand := (Index := DataRecord#StartType );
            CraterFillTime : UIntAsyncCommand := (Index := DataRecord#CraterFillTime);
            BurnBackTime : UIntAsyncCommand := (Index := DataRecord#BurnBackTime);
            LwasNoOfStarts : UIntAsyncCommand := (Index := DataRecord#LwasNoOfStarts);
            LwasTimeout : UIntAsyncCommand := (Index := DataRecord#LwasTimeout);
            CableArea : UIntAsyncCommand := (Index := DataRecord#CableArea);
            CableLength : UIntAsyncCommand := (Index := DataRecord#CableLength);
            GetWireDimensions : UIntAsyncCommand := (Index := DataRecord#GetWireDimensions);
            GetWireTypes : UIntAsyncCommand := (Index := DataRecord#GetWireTypes);
            MeasureValueFrequency : UIntAsyncCommand := (Index := DataRecord#MeasureValueFrequency);
            MaxOcv : UIntAsyncCommand := (Index := DataRecord#MaxOcv);
            ParallelPowerSources : UIntAsyncCommand := (Index := DataRecord#ParallelPowerSources);
            AcSyncMaster : UIntAsyncCommand := (Index := DataRecord#AcSyncMaster);
            CoupleId : UIntAsyncCommand := (Index := DataRecord#CoupleId);
            PairParallelCouple : UIntAsyncCommand := (Index := DataRecord#PairParallelCouple);
            MeasureValueFilter : UIntAsyncCommand := (Index := DataRecord#MeasureValueFilter);
            TandemRole : UIntAsyncCommand := (Index := DataRecord#TandemRole);
            CreepStart : UIntAsyncCommand := (Index := DataRecord#CreepStart);
            CreepSpeed : UIntAsyncCommand := (Index := DataRecord#CreepSpeed);
            MaxTravelSpeed : UIntAsyncCommand := (Index := DataRecord#MaxTravelSpeed);
            TravelControl : UIntAsyncCommand := (Index := DataRecord#TravelControl);
            TravelMotorDrive : UIntAsyncCommand := (Index := DataRecord#TravelMotorDrive);
            WireMotorScaleFactor1 : UIntAsyncCommand := (Index := DataRecord#WireMotorScaleFactor1);
            WireMotorScaleFactor2 : UIntAsyncCommand := (Index := DataRecord#WireMotorScaleFactor2);
            MaxWireMotorCurrent : UIntAsyncCommand := (Index := DataRecord#MaxWireMotorCurrent);
            ConnectedUnits : UDIntAsyncCommand := (Index := DataRecord#ConnectedUnits);
            NodeInformation : NodeInformationAsyncCommand := (Index := DataRecord#NodeInformation);
            Can2NodeId : UIntAsyncCommand := (Index := DataRecord#Can2NodeId);
            GetWeldingSystem : UIntAsyncCommand := (Index := DataRecord#GetWeldingSystem);
            JogWireFeedSpeed : UIntAsyncCommand := (Index := DataRecord#WireJogLowSpeed);
            JogWireFeedHighSpeed : UIntAsyncCommand := (Index := DataRecord#WireJogHighSpeed);
        END_VAR
    END_CLASS

    CLASS UIntAsyncCommand EXTENDS AsyncCommand
        VAR PUBLIC
            Value : UINT := UINT#0;
        END_VAR

        METHOD PUBLIC OVERRIDE ValueAsBytes
            VAR_INPUT
                buffer : REF_TO ARRAY[*] OF BYTE;
            END_VAR

            buffer^[0] := Value.%B1;
            buffer^[1] := Value.%B0;
        END_METHOD

        METHOD PUBLIC OVERRIDE ValueFromBytes
            VAR_INPUT
                buffer : REF_TO ARRAY[*] OF BYTE;
            END_VAR

            Value.%B1 := buffer^[0];
            Value.%B0 := buffer^[1];
        END_METHOD

        METHOD PUBLIC OVERRIDE GetSize : UINT
            GetSize := UINT#2;
        END_METHOD
    END_CLASS

    CLASS UDIntAsyncCommand EXTENDS AsyncCommand
        VAR PUBLIC
            Value : UDINT := UDINT#0;
        END_VAR

        METHOD PUBLIC OVERRIDE ValueAsBytes
            VAR_INPUT
                buffer : REF_TO ARRAY[*] OF BYTE;
            END_VAR

            buffer^[0] := Value.%B1;
            buffer^[1] := Value.%B0;
            buffer^[2] := Value.%B3;
            buffer^[3] := Value.%B2;
        END_METHOD

        METHOD PUBLIC OVERRIDE ValueFromBytes
            VAR_INPUT
                buffer : REF_TO ARRAY[*] OF BYTE;
            END_VAR

            Value.%B1 := buffer^[0];
            Value.%B0 := buffer^[1];
            Value.%B3 := buffer^[2];
            Value.%B2 := buffer^[3];
        END_METHOD

        METHOD PUBLIC OVERRIDE GetSize : UINT
            GetSize := UINT#4;
        END_METHOD
    END_CLASS

    CLASS RealAsyncCommand EXTENDS AsyncCommand
        VAR PUBLIC
            Value : REAL := REAL#0.0;
        END_VAR

        METHOD PUBLIC OVERRIDE ValueAsBytes
            VAR_INPUT
                buffer : REF_TO ARRAY[*] OF BYTE;
            END_VAR

            VAR_TEMP
                _value : DWORD;
            END_VAR

            _value := TO_DWORD(Value);

            buffer^[0] := _value.%B1;
            buffer^[1] := _value.%B0;
            buffer^[2] := _value.%B3;
            buffer^[3] := _value.%B2;
        END_METHOD

        METHOD PUBLIC OVERRIDE ValueFromBytes
            VAR_INPUT
                buffer : REF_TO ARRAY[*] OF BYTE;
            END_VAR

            VAR_TEMP
                _value : DWORD;
            END_VAR

            _value.%B1 := buffer^[0];
            _value.%B0 := buffer^[1];
            _value.%B3 := buffer^[2];
            _value.%B2 := buffer^[3];

            Value := TO_REAL(_value);
        END_METHOD

        METHOD PUBLIC OVERRIDE GetSize : UINT
            GetSize := UINT#4;
        END_METHOD
    END_CLASS

    /// Async command that fetches the information of a node
    /// This command is a bit special. When used to write it will
    /// send the provided id, and when used to read it will populate the
    /// Value variable.
    CLASS NodeInformationAsyncCommand EXTENDS AsyncCommand
        VAR PUBLIC
            Id : UINT;
            Value : NodeInformation;
        END_VAR

        METHOD PUBLIC OVERRIDE ValueAsBytes
            VAR_INPUT
                buffer : REF_TO ARRAY[*] OF BYTE;
            END_VAR

            buffer^[0] := Id.%B1;
            buffer^[1] := Id.%B0;
        END_METHOD

        METHOD PUBLIC OVERRIDE ValueFromBytes
            VAR_INPUT
                buffer : REF_TO ARRAY[*] OF BYTE;
            END_VAR

            VAR_TEMP
                Version : UINT;
                SubVersion : UINT;
                DeviceType : UINT;
                MachineId : UINT;
            END_VAR

            Version.%B1 := buffer^[0];
            Version.%B0 := buffer^[1];
            SubVersion.%B1 := buffer^[2];
            SubVersion.%B0 := buffer^[3];
            DeviceType.%B1 := buffer^[4];
            DeviceType.%B0 := buffer^[5];
            MachineId.%B1 := buffer^[6];
            MachineId.%B0 := buffer^[7];

            Value.Version := Version;
            Value.SubVersion := TO_CHAR(TO_BYTE(SubVersion));
            Value.DeviceType := DeviceType;
            Value.MachineId := MachineId;
        END_METHOD

        METHOD PUBLIC OVERRIDE GetSize : UINT
            GetSize := UINT#8;
        END_METHOD
    END_CLASS

END_NAMESPACE

(* ---- AsyncInterface.st ---- *)
USING Esab.Utils.Alarming;
USING Esab.Utils.Collections;

USING Siemens.Simatic.S71500.DistributedIO;
USING Siemens.Simatic.S71500.Alarming;

NAMESPACE Esab.WeldSystem.PowerSources

    CLASS PUBLIC AsyncInterface IMPLEMENTS IAsyncInterface
        VAR PRIVATE
            _reader : IAsyncReader;
            _writer : IAsyncWriter;
            _invalidCommandTypeAlarm : IAlarm;
            _poppedNullCommandAlarm : IAlarm;
            _invalidCommandAlarm : IAlarm;

            _commandQueue : LinkedList;
            _currentCommand : REF_TO AsyncCommand := NULL;
            _listener : IAsyncCommandListener := NULL;
            _successfullyExecutedCommandsCounter : UINT;
            _executedCommandsCounter : UINT;
            _executingCommandCounter : UINT;
            _nextCommandCounter : UINT;
            _busy : BOOL;
        END_VAR

        VAR PRIVATE
            {S7.Alarm = NoAck, "Async command interface not initialized."}
            _initializationAlarm : ProgramAlarm;
        END_VAR

        METHOD PUBLIC Setup
            VAR_INPUT
                reader : IAsyncReader;
                writer : IAsyncWriter;
                invalidCommandTypeAlarm : IAlarm;
                poppedNullCommandAlarm : IAlarm;
                invalidCommandAlarm : IAlarm;
            END_VAR

            _reader := reader;
            _writer := writer;
            _invalidCommandTypeAlarm := invalidCommandTypeAlarm;
            _poppedNullCommandAlarm := poppedNullCommandAlarm;
            _invalidCommandAlarm := invalidCommandAlarm;
        END_METHOD

        METHOD PUBLIC IsInitialized : BOOL
            VAR_TEMP
                initialized : BOOL := FALSE;
            END_VAR

            initialized :=
                _reader <> NULL AND
                _writer <> NULL AND
                _invalidCommandTypeAlarm <> NULL AND
                _poppedNullCommandAlarm <> NULL AND
                _invalidCommandAlarm <> Null;

            _initializationAlarm(SIG := NOT initialized);

            IsInitialized := initialized;
        END_METHOD

        METHOD PUBLIC Execute
            VAR_TEMP
                _linkedListItem : REF_TO LinkedListItem;
            END_VAR

            IF NOT THIS.IsInitialized() THEN
                RETURN;
            END_IF;

            IF _commandQueue.Size() > 0 AND _currentCommand = NULL THEN
                    _linkedListItem := _commandQueue.PopHead();
                    _currentCommand ?= _linkedListItem;

                    _nextCommandCounter := _nextCommandCounter + UINT#1;

                    _poppedNullCommandAlarm.Execute(SIG := _linkedListItem = NULL);
                    _invalidCommandAlarm.Execute(SIG := _linkedListItem <> NULL AND _currentCommand = NULL);
                    IF _currentCommand <> NULL THEN
                        _invalidCommandTypeAlarm.Execute(SIG := NOT (_currentCommand^.GetType() = CommandType#Read OR _currentCommand^.GetType() = CommandType#Write));
                        CASE _currentCommand^.GetType() OF
                            CommandType#Read:
                                _reader.SetCommand(_currentCommand);
                            CommandType#Write:
                                _writer.SetCommand(_currentCommand);
                        ELSE
                            _currentCommand := NULL;
                        END_CASE;
                    END_IF;
            ELSIF _currentCommand = NULL AND NOT (_reader.IsBusy() OR _writer.IsBusy()) THEN
                _reader.SetCommand(NULL);
                _writer.SetCommand(NULL);
            END_IF;

            _busy := _currentCommand <> NULL;

            _reader.Execute();
            _writer.Execute();

            IF _reader.IsBusy() OR _writer.IsBusy() THEN
                _executingCommandCounter := _executingCommandCounter + UINT#1;
            END_IF;

            IF _reader.IsDone() OR _writer.IsDone() THEN
                IF _listener <> NULL THEN
                    _listener.AsyncCommandCallback(_currentCommand, CommandStatus#Success);
                END_IF;
                _currentCommand^.Callback(CommandStatus#Success);

                _executedCommandsCounter := _executedCommandsCounter + UINT#1;
                _successfullyExecutedCommandsCounter := _successfullyExecutedCommandsCounter + UINT#1;

                THIS.Reset();
            END_IF;

            IF _reader.HasError() OR _writer.HasError() THEN
                IF _listener <> NULL THEN
                    _listener.AsyncCommandCallback(_currentCommand, CommandStatus#Error);
                END_IF;
                _currentCommand^.Callback(CommandStatus#Error);
                _executedCommandsCounter := _executedCommandsCounter + UINT#1;

                THIS.Reset();
            END_IF;
        END_METHOD

        METHOD PUBLIC Reset
            _currentCommand := NULL;

            _reader.SetCommand(NULL);
            _writer.SetCommand(NULL);

            _reader.Execute();
            _writer.Execute();
        END_METHOD

        METHOD PUBLIC WriteCommand
            VAR_INPUT
                command : REF_TO AsyncCommand;
            END_VAR

            IF _commandQueue.Append(command) THEN
                command^.SetWrite();
            END_IF;
        END_METHOD

        METHOD PUBLIC ReadCommand
            VAR_INPUT
                command : REF_TO AsyncCommand;
            END_VAR

            IF _commandQueue.Append(command) THEN
                command^.SetRead();
            END_IF;
        END_METHOD

        METHOD PUBLIC FlushCommandQueue
            _commandQueue.Clear();
        END_METHOD

        METHOD PUBLIC CurrentCommand : REF_TO AsyncCommand
            CurrentCommand := _currentCommand;
        END_METHOD

        METHOD PUBLIC IsIdle : BOOL
            IsIdle := _commandQueue.Empty() AND _currentCommand = NULL AND NOT _reader.IsBusy() AND NOT _writer.IsBusy();
        END_METHOD

        METHOD PUBLIC SetListener
            VAR_INPUT
                handler : IAsyncCommandListener;
            END_VAR

            _listener := handler;
        END_METHOD
    END_CLASS

    CLASS AsyncReader IMPLEMENTS IAsyncReader
        VAR PUBLIC
            HwId : WORD;
            ErrorAlarm: IAlarm;
        END_VAR

        VAR PRIVATE
            _reader : ReadRecord;
            _command : REF_TO AsyncCommand;

            _valid : BOOL;
            _error : BOOL;
            _busy : BOOL;

            _record : ARRAY[0..10] OF BYTE;
        END_VAR

        METHOD PUBLIC Execute
            VAR_TEMP
                status : DWORD := DWORD#0;
                request : BOOL := FALSE;
                length : UINT := UINT#0;
                index : DINT := DINT#0;
                maxLength : UINT := UINT#0;
            END_VAR

            IF _command <> NULL THEN
                request := TRUE;
                index := _command^.GetIndex();
                maxLength := _command^.GetSize();
            ELSE
                request := FALSE;
            END_IF;

            _reader(
                request := request,
                id := HwId,
                index := index,
                maxLength := length,
                record := _record,
                valid => _valid,
                busy => _busy,
                error => _error,
                status => status,
                length => length
            );

            IF _command <> NULL AND _valid THEN
                _command^.ValueFromBytes(REF(_record));
            END_IF;

            ErrorAlarm.Execute(SIG := _error, SD_1 := pass(status));
        END_METHOD

        METHOD PUBLIC SetCommand
            VAR_INPUT
                command : REF_TO AsyncCommand;
            END_VAR

            _command := command;
        END_METHOD

        METHOD PUBLIC IsDone : BOOL
            IsDone := _valid;
        END_METHOD

        METHOD PUBLIC IsBusy : BOOL
            IsBusy := _busy;
        END_METHOD

        METHOD PUBLIC HasError : BOOL
            HasError := _error;
        END_METHOD
    END_CLASS

    CLASS AsyncWriter IMPLEMENTS IAsyncWriter
        VAR PUBLIC
            HwId : WORD;
            ErrorAlarm : IAlarm;
        END_VAR

        VAR PRIVATE
            _writer : WriteRecord;
            _command : REF_TO AsyncCommand;

            _valid : BOOL;
            _error : BOOL;
            _busy : BOOL;

            _record : ARRAY[0..10] OF BYTE;
        END_VAR

        METHOD PUBLIC Execute
            VAR_TEMP
                status : DWORD := DWORD#0;
                request : BOOL := FALSE;
                length : UINT := UINT#0;
                index : DINT := DINT#0;
                maxLength : UINT := UINT#0;
            END_VAR

            IF _command <> NULL THEN
                request := TRUE;
                index := _command^.GetIndex();
                maxLength := _command^.GetSize();
                _command^.ValueAsBytes(REF(_record));
            ELSE
                request := FALSE;
            END_IF;

            _writer(
                request := request,
                id := HwId,
                index := index,
                length := length,
                record := _record,
                done => _valid,
                busy => _busy,
                error => _error,
                status => status
            );

            ErrorAlarm.Execute(SIG := _error, SD_1 := pass(status));
        END_METHOD

        METHOD PUBLIC SetCommand
            VAR_INPUT
                command : REF_TO AsyncCommand;
            END_VAR

            _command := command;
        END_METHOD

        METHOD PUBLIC IsDone : BOOL
            IsDone := _valid;
        END_METHOD

        METHOD PUBLIC IsBusy : BOOL
            IsBusy := _busy;
        END_METHOD

        METHOD PUBLIC HasError : BOOL
            HasError := _error;
        END_METHOD
    END_CLASS

    INTERFACE IAsyncInterface
        /// Cyclic execute.
        METHOD Execute
        END_METHOD

        /// Resets the internal state (does NOT flush the command queue)
        METHOD Reset
        END_METHOD

        /// Adds a write command to the execution queue.
        METHOD WriteCommand
            VAR_INPUT
                command : REF_TO AsyncCommand;
            END_VAR
        END_METHOD

        /// Adds a write command to the execution queue.
        METHOD ReadCommand
            VAR_INPUT
                command : REF_TO AsyncCommand;
            END_VAR
        END_METHOD

        /// Clears the command queue (this will NOT abort any running commands).
        METHOD FlushCommandQueue
        END_METHOD

        /// Returns a reference to the current command
        METHOD CurrentCommand : REF_TO AsyncCommand
        END_METHOD

        /// Returns TRUE if this async interface is idle (i.e. no commands in queue)
        METHOD IsIdle : BOOL
        END_METHOD

        METHOD SetListener
            VAR_INPUT
                handler : IAsyncCommandListener;
            END_VAR
        END_METHOD
    END_INTERFACE

    CLASS ABSTRACT AsyncCommand EXTENDS LinkedListItem IMPLEMENTS IAsyncCommand
        VAR PUBLIC
            CommandType : CommandType := CommandType#Invalid;
            Index : DataRecord := DataRecord#Invalid;
        END_VAR

        VAR PRIVATE
            _callback_listener : IAsyncCommandListener := NULL;
        END_VAR

        METHOD PUBLIC GetIndex : DataRecord
            GetIndex := Index;
        END_METHOD

        METHOD PUBLIC ABSTRACT ValueAsBytes
            VAR_INPUT
                buffer : REF_TO ARRAY[*] OF BYTE;
            END_VAR
        END_METHOD

        METHOD PUBLIC ABSTRACT ValueFromBytes
            VAR_INPUT
                buffer : REF_TO ARRAY[*] OF BYTE;
            END_VAR
        END_METHOD

        METHOD PUBLIC ABSTRACT GetSize : UINT
        END_METHOD

        METHOD PUBLIC SetWrite
            CommandType := CommandType#Write;
        END_METHOD

        METHOD PUBLIC SetRead
            CommandType := CommandType#Read;
        END_METHOD

        METHOD PUBLIC GetType : CommandType
            GetType := CommandType;
        END_METHOD

        METHOD PUBLIC SetListener
            VAR_INPUT
                Listener : IAsyncCommandListener;
            END_VAR
            _callback_listener := Listener;
        END_METHOD

        METHOD PUBLIC Callback
            VAR_INPUT
                status : CommandStatus;
            END_VAR
            IF _callback_listener <> NULL THEN
                _callback_listener.AsyncCommandCallback(REF(THIS), status);
            END_IF;
        END_METHOD
    END_CLASS

    INTERFACE IAsyncCommand
        /// The data record to be read/written.
        METHOD GetIndex : DataRecord
        END_METHOD

        /// Writes the command data into a buffer
        METHOD ValueAsBytes
            VAR_INPUT
                buffer : REF_TO ARRAY[*] OF BYTE;
            END_VAR
        END_METHOD

        /// Reads a buffer and converts it into the command value
        METHOD ValueFromBytes
            VAR_INPUT
                buffer : REF_TO ARRAY[*] OF BYTE;
            END_VAR
        END_METHOD

        /// The expected size of the data in bytes.
        METHOD GetSize : UINT
        END_METHOD

        /// Set the type of this command to write
        METHOD SetWrite
        END_METHOD

        /// Set the type of this command to read
        METHOD SetRead
        END_METHOD

        /// The type of command (read or write).
        METHOD GetType : CommandType
        END_METHOD

        /// Listen for when the command finishes.
        METHOD SetListener
            VAR_INPUT
                Listener : IAsyncCommandListener;
            END_VAR
        END_METHOD

        /// Callback the command once finished to the listener.
        METHOD Callback
            VAR_INPUT
                status : CommandStatus;
            END_VAR
        END_METHOD
    END_INTERFACE

    INTERFACE IAsyncCommandListener
        METHOD AsyncCommandCallback
            VAR_INPUT
                command : REF_TO AsyncCommand;
                status : CommandStatus;
            END_VAR
        END_METHOD
    END_INTERFACE

    INTERFACE IAsyncWriter

        /// Cyclic execute.
        METHOD Execute
        END_METHOD

        /// Sets the command to be executed by the writer
        METHOD SetCommand
            VAR_INPUT
                command : REF_TO AsyncCommand;
            END_VAR
        END_METHOD

        /// Returns TRUE if the write operation was successful.
        METHOD IsDone : BOOL
        END_METHOD

        /// Returns TRUE if the write operation is in progress.
        METHOD IsBusy : BOOL
        END_METHOD

        /// Returns TRUE if an error occured during write.
        METHOD HasError : BOOL
        END_METHOD

    END_INTERFACE

    INTERFACE IAsyncReader

        /// Cyclic execute.
        METHOD Execute
        END_METHOD

        /// Sets the command to be executed by the reader
        METHOD SetCommand
            VAR_INPUT
                command : REF_TO AsyncCommand;
            END_VAR
        END_METHOD

        /// Returns TRUE if the read operation was successful.
        METHOD IsDone : BOOL
        END_METHOD

        /// Returns TRUE if the read operation is in progress.
        METHOD IsBusy : BOOL
        END_METHOD

        /// Returns TRUE if an error occured during read.
        METHOD HasError : BOOL
        END_METHOD

    END_INTERFACE

    TYPE
        CommandType : INT(
            Invalid := INT#-1,
            Read := INT#0,
            Write := INT#1
        ) := Invalid;

        CommandStatus : INT(
            Invalid := -1,
            Success := 0,
            Error := 1
        ) := Error;

        DataRecord : DINT(
            Invalid := DINT#-1,
            WeldProcess := DINT#1,
            WeldMethod := DINT#2,
            RegulationType := DINT#3,
            WireType := DINT#4,
            WireDimension := DINT#5,
            Voltage := DINT#6,
            Current := DINT#7,
            StartType := DINT#8,
            CraterFillTime := DINT#9,
            BurnBackTime := DINT#10,
            RegulationDynamics := DINT#11,
            RegulationInductance := DINT#12,
            AcFrequency := DINT#13,
            AcBalance := DINT#14,
            AcOffset := DINT#15,
            AcPhaseShift := DINT#16,
            StartAdjust := DINT#17,
            WireSpeed := DINT#18,
            TravelSpeed := DINT#19,
            IceWireSpeedPercentage := DINT#21,
            LwasNoOfStarts := DINT#22,
            LwasTimeout := DINT#23,
            CableArea := DINT#30,
            CableLength := DINT#31,
            GetWireDimensions := DINT#32,
            GetWireTypes := DINT#33,
            MeasureValueFrequency := DINT#34,
            MaxOcv := DINT#35,
            ParallelPowerSources := DINT#36,
            AcSyncMaster := DINT#37,
            CoupleId := DINT#38,
            PairParallelCouple := DINT#39,
            MeasureValueFilter := DINT#40,
            TandemRole := DINT#41,
            CreepStart := DINT#43,
            CreepSpeed := DINT#44,
            MaxTravelSpeed := DINT#45,
            TravelControl := DINT#46,
            TravelMotorDrive := DINT#47,
            WireMotorScaleFactor1 := DINT#48,
            WireMotorScaleFactor2 := DINT#49,
            WireJogLowSpeed := DINT#50,
            WireJogHighSpeed := DINT#51,
            IceActive := DINT#55,
            IceStartDelay := DINT#56,
            IceWireMotorScaleFactor1 := DINT#57,
            IceWireMotorScaleFactor2 := DINT#58,
            IceWireJogLowSpeed := DINT#59,
            IceWireJogHighSpeed := DINT#60,
            IceLicenseRemainingTime := DINT#61,
            MaxWireMotorCurrent := DINT#63,
            LanguageSelection := DINT#100,
            ConnectedUnits := DINT#107,
            NodeInformation := DINT#108,
            GetWeldingSystem := DINT#109,
            ErrorMessage := DINT#112,
            ErrorDeviceType := DINT#113,
            Can2NodeId := DINT#115
        ) := Invalid;

        NodeInformation : STRUCT
            Connected : BOOL := FALSE;
            Version : UINT := UINT#0;
            SubVersion : CHAR := CHAR#0;
            DeviceType : DeviceType := DeviceType#Invalid;
            MachineId : UINT := UINT#0;
        END_STRUCT;

        DeviceType : UINT(
            Invalid := UINT#99,
            WeldDataUnit := UINT#0,
            PowerSource := UINT#2,
            MotorControl := UINT#6
        ) := Invalid;

        WeldSystemType : UINT(
            LafTaf := UINT#0,
            Aristo1000 := UINT#1
        );
    END_TYPE

END_NAMESPACE
